// TIA Portal V19 program export: 1 tag tables, 6 data types, 2 data blocks, 8 code blocks (in call order from the OBs), 5 instance data blocks

VAR_GLOBAL   // PLC tag table "Default tag table"
   Tag_1 AT %M0.5 : Bool;
   Clock_Byte AT %MB0 : Byte;
   Clock_10Hz AT %M0.0 : Bool;
   Clock_5Hz AT %M0.1 : Bool;
   "Clock_2.5Hz" AT %M0.2 : Bool;
   Clock_2Hz AT %M0.3 : Bool;
   "Clock_1.25Hz" AT %M0.4 : Bool;
   Clock_1Hz AT %M0.5 : Bool;
   "Clock_0.625Hz" AT %M0.6 : Bool;
   "Clock_0.5Hz" AT %M0.7 : Bool;
   VibSensor01 AT %I100.0 : "PII - BCM R15E-001-DI00-01,5-S4";
   VibSensor02 AT %I124.0 : "PII - BCM R15E-001-DI00-01,5-S4";
   VibSensor03 AT %I148.0 : "PII - BCM R15E-001-DI00-01,5-S4";
   TempHumidSensor01 AT %I172.0 : "PII - CSS 01411.2-xx";
   OilContaminationSensor01 AT %I184.0 : "PII - BCI24-DH367-1D1A-4";
   AirFlowSensor01 AT %I194.0 : "PII - AS5-AF2-FLX-G100";
END_VAR

TYPE "PII - AS5-AF2-FLX-G100"
   STRUCT
      "Process Data In - Mass Flow Rate" : Real;
      "Process Data In - Flow Velocity" : Real;
      "Process Data In - Volume" : Real;
      "Process Data In - Volumetric Flow Rate" : Real;
      "Process Data In - Mass" : Real;
      "Process Data In - Energy" : Real;
      "Process Data In - Temperature" : Real;
      "Process Data In - Pressure" : Real;
      "Port qualifier" : Byte;
   END_STRUCT;
END_TYPE

TYPE "PII - BCI24-DH367-1D1A-4"
   STRUCT
      "Process Data In - Switching output 1" : Bool;
      "Reserved Bit" : Bool;
      "Reserved Bit_1" : Bool;
      "Reserved Bit_2" : Bool;
      "Reserved Bit_3" : Bool;
      "Reserved Bit_4" : Bool;
      "Reserved Bit_5" : Bool;
      "Reserved Bit_6" : Bool;
      "Reserved Byte" : Bool;
      "Process Data In - Pressure" : Word;
      "Reserved Byte_1" : Bool;
      "Reserved Byte_2" : Bool;
      "Reserved Byte_3" : Bool;
      "Reserved Byte_4" : Bool;
      "Reserved Byte_5" : Bool;
      "Reserved Byte_6" : Bool;
      "Reserved Byte_7" : Bool;
      "Reserved Byte_8" : Bool;
      "Reserved Byte_9" : Bool;
      "Reserved Byte_10" : Bool;
      "Reserved Byte_11" : Bool;
      "Reserved Byte_12" : Bool;
      "Reserved Byte_13" : Bool;
      "Reserved Byte_14" : Bool;
      "Reserved Byte_15" : Bool;
      "Reserved Byte_16" : Bool;
      "Reserved Byte_17" : Bool;
      "Reserved Byte_18" : Bool;
      "Reserved Byte_19" : Bool;
      "Reserved Byte_20" : Bool;
      "Reserved Byte_21" : Bool;
      "Reserved Byte_22" : Bool;
      "Reserved Byte_23" : Bool;
      "Reserved Byte_24" : Bool;
      "Reserved Byte_25" : Bool;
      "Reserved Byte_26" : Bool;
      "Reserved Byte_27" : Bool;
      "Reserved Byte_28" : Bool;
      "Port qualifier" : Byte;
   END_STRUCT;
END_TYPE

TYPE "PII - BCM R15E-001-DI00-01,5-S4"
   STRUCT
      "Vibration Acceleration - Vibration Acceleration RMS a-RMS X" : Real;
      "Vibration Acceleration - Vibration Acceleration RMS a-RMS Y" : Real;
      "Vibration Acceleration - Vibration Acceleration RMS a-RMS Z" : Real;
      "Vibration Acceleration - Contact Temperature Contact Temperature" : Real;
      "Vibration Acceleration - Status Bits Main-Alarm a-RMS Magnitude Status" : Bool;
      "Vibration Acceleration - Status Bits Pre-Alarm a-RMS Magnitude Status" : Bool;
      "Vibration Acceleration - Status Bits Main-Alarm a-RMS Z Status" : Bool;
      "Vibration Acceleration - Status Bits Pre-Alarm a-RMS Z Status" : Bool;
      "Vibration Acceleration - Status Bits Main-Alarm a-RMS Y Status" : Bool;
      "Vibration Acceleration - Status Bits Pre-Alarm a-RMS Y Status" : Bool;
      "Vibration Acceleration - Status Bits Main-Alarm a-RMS X Status" : Bool;
      "Vibration Acceleration - Status Bits Pre-Alarm a-RMS X Status" : Bool;
      "Vibration Acceleration - Status Bits Main-Alarm v-RMS Magnitude Status" : Bool;
      "Vibration Acceleration - Status Bits Pre-Alarm v-RMS Magnitude Status" : Bool;
      "Vibration Acceleration - Status Bits Main-Alarm v-RMS Z Status" : Bool;
      "Vibration Acceleration - Status Bits Pre-Alarm v-RMS Z Status" : Bool;
      "Vibration Acceleration - Status Bits Main-Alarm v-RMS Y Status" : Bool;
      "Vibration Acceleration - Status Bits Pre-Alarm v-RMS Y Status" : Bool;
      "Vibration Acceleration - Status Bits Main-Alarm v-RMS X Status" : Bool;
      "Vibration Acceleration - Status Bits Pre-Alarm v-RMS X Status" : Bool;
      "Vibration Acceleration - Status Bits Reserved" : Bool;
      "Vibration Acceleration - Status Bits Reserved_1" : Bool;
      "Vibration Acceleration - Status Bits Reserved_2" : Bool;
      "Vibration Acceleration - Status Bits Vibration Severity Zone D" : Bool;
      "Vibration Acceleration - Status Bits Vibration Severity Zone C" : Bool;
      "Vibration Acceleration - Status Bits Vibration Severity Zone B" : Bool;
      "Vibration Acceleration - Status Bits Vibration Severity Zone A" : Bool;
      "Vibration Acceleration - Status Bits Reserved_3" : Bool;
      "Vibration Acceleration - Status Bits Reserved_4" : Bool;
      "Vibration Acceleration - Status Bits Reserved_5" : Bool;
      "Vibration Acceleration - Status Bits Reserved_6" : Bool;
      "Vibration Acceleration - Status Bits Reserved_7" : Bool;
      "Vibration Acceleration - Status Bits Reserved_8" : Bool;
      "Vibration Acceleration - Status Bits Reserved_9" : Bool;
      "Vibration Acceleration - Status Bits Contact Temperature Upper Alarm Status" : Bool;
      "Vibration Acceleration - Status Bits Contact Temperature Lower Alarm Status" : Bool;
      "Reserved Byte" : Bool;
      "Reserved Byte_1" : Bool;
      "Reserved Byte_2" : Bool;
      "Reserved Byte_3" : Bool;
      "Reserved Byte_4" : Bool;
      "Reserved Byte_5" : Bool;
      "Reserved Byte_6" : Bool;
      "Reserved Byte_7" : Bool;
      "Reserved Byte_8" : Bool;
      "Reserved Byte_9" : Bool;
      "Reserved Byte_10" : Bool;
      "Reserved Byte_11" : Bool;
      "Port qualifier" : Byte;
   END_STRUCT;
END_TYPE

TYPE "PII - CSS 01411.2-xx"
   STRUCT
      "Process Data Inputs - Temperature" : Int;
      "Process Data Inputs - Temperature Alarm High" : Bool;
      "Process Data Inputs - Temperature Range High" : Bool;
      "Process Data Inputs - Temperature Range Low" : Bool;
      "Process Data Inputs - Temperature Alarm Low" : Bool;
      "Reserved Bit" : Bool;
      "Reserved Bit_1" : Bool;
      "Reserved Bit_2" : Bool;
      "Reserved Bit_3" : Bool;
      "Process Data Inputs - Humidity" : Int;
      "Process Data Inputs - Humidity Alarm High" : Bool;
      "Process Data Inputs - Humidity Range High" : Bool;
      "Process Data Inputs - Humidity Range Low" : Bool;
      "Process Data Inputs - Humidity Alarm Low" : Bool;
      "Reserved Bit_4" : Bool;
      "Reserved Bit_5" : Bool;
      "Reserved Bit_6" : Bool;
      "Reserved Bit_7" : Bool;
      "Reserved Byte" : Bool;
      "Reserved Byte_1" : Bool;
      "Reserved Byte_2" : Bool;
      "Reserved Byte_3" : Bool;
      "Reserved Byte_4" : Bool;
      "Reserved Byte_5" : Bool;
      "Reserved Byte_6" : Bool;
      "Reserved Byte_7" : Bool;
      "Reserved Byte_8" : Bool;
      "Reserved Byte_9" : Bool;
      "Reserved Byte_10" : Bool;
      "Reserved Byte_11" : Bool;
      "Reserved Byte_12" : Bool;
      "Reserved Byte_13" : Bool;
      "Reserved Byte_14" : Bool;
      "Reserved Byte_15" : Bool;
      "Reserved Byte_16" : Bool;
      "Reserved Byte_17" : Bool;
      "Reserved Byte_18" : Bool;
      "Reserved Byte_19" : Bool;
      "Reserved Byte_20" : Bool;
      "Reserved Byte_21" : Bool;
      "Reserved Byte_22" : Bool;
      "Reserved Byte_23" : Bool;
      "Reserved Byte_24" : Bool;
      "Reserved Byte_25" : Bool;
      "Port qualifier" : Byte;
   END_STRUCT;
END_TYPE

TYPE "typeSimSensors"
   STRUCT
      Sensors : Struct
         Sensor11 : Real;   // Machine 001 / Sensor 001
         Sensor12 : Real;   // Machine 001 / Sensor 002
         Sensor13 : Real;   // Machine 001 / Sensor 003
         Sensor14 : Real;   // Machine 001 / Sensor 004
         Sensor21 : Real;   // Machine 002 / Sensor 001
         Sensor22 : Real;   // Machine 002 / Sensor 002
         Sensor23 : Real;   // Machine 002 / Sensor 003
         Sensor24 : Real;   // Machine 002 / Sensor 004
      END_STRUCT;
   END_STRUCT;
END_TYPE

TYPE "typeSimStates"
   STRUCT
      States : Struct
         State11 : UInt;   // Machine 1 / State 1
         State12 : UInt;   // Machine 1 / State 2
         State13 : UInt;   // Machine 1 / State 3
         State14 : UInt;   // Machine 1 / State 4
         State21 : UInt;   // Machine 2 / State 1
         State22 : UInt;   // Machine 2 / State 2
         State23 : UInt;   // Machine 2 / State 3
         State24 : UInt;   // Machine 2 / State 4
      END_STRUCT;
   END_STRUCT;
END_TYPE

DATA_BLOCK "GlobalConst_DB"   // DB8
{ S7_Optimized_Access := 'TRUE' }
// stored: MemoryReserve 100
   VAR
      mqtt_host_address : String := '192.168.1.165';
      mqtt_port : UInt := 1883;
      mqtt_username : WString := WSTRING#'mqttbroker';
      mqtt_password : WString := WSTRING#'IoT@2023';
   END_VAR
BEGIN
END_DATA_BLOCK

DATA_BLOCK "GlobalData"   // DB6
{ S7_Optimized_Access := 'TRUE' }
// stored: MemoryReserve 100
   VAR
      UnixTimestamp : DInt;
      SensorsSimulation : "typeSimSensors";
      StatesSimulation { S7_SetPoint := 'True'} : "typeSimStates";
   END_VAR
BEGIN
END_DATA_BLOCK

ORGANIZATION_BLOCK "Main"   // OB1, LAD, ProgramCycle
TITLE = "Main Program Sweep (Cycle)"
{ S7_Optimized_Access := 'TRUE' }
// stored: SetENOAutomatically false
   VAR_INPUT
      Initial_Call : Bool;   // Initial call of this OB
      Remanence : Bool;   // =True, if remanent data are available
   END_VAR
BEGIN

REGION Network 1: Sensor / States simulation
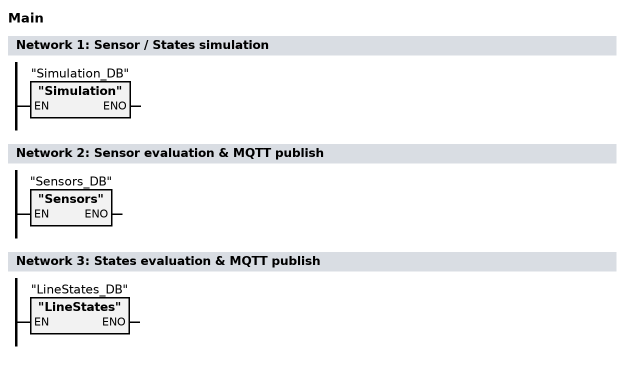
   RUNG wire#powerrail
      "Simulation_DB"()
   END_RUNG
   // the same network as SCL:
   "Simulation_DB"();   // "Simulation"
END_REGION

REGION Network 2: Sensor evaluation & MQTT publish
   RUNG wire#powerrail
      "Sensors_DB"()
   END_RUNG
   // the same network as SCL:
   "Sensors_DB"();   // "Sensors"
END_REGION

REGION Network 3: States evaluation & MQTT publish
   RUNG wire#powerrail
      "LineStates_DB"()
   END_RUNG
   // the same network as SCL:
   "LineStates_DB"();   // "LineStates"
END_REGION
END_ORGANIZATION_BLOCK

FUNCTION_BLOCK "Simulation"   // FB1, LAD
{ S7_Optimized_Access := 'TRUE' }
// stored: MemoryReserve 100, SetENOAutomatically false
   VAR
      LGF_Error : Array[1..10] of Bool;
      LGF_Status : Array[1..10] of Word;
      RetValReal : Real;
   END_VAR
   VAR_TEMP
      RndDIntStatus : Array[1..10] of Word;
      RndRealStatus : Array[1..10] of Word;
   END_VAR
   VAR_TEMP   // added for the SCL form of the ladder/FBD networks
      _w1 : Bool;
      _w2 : Bool;
      _w3 : Bool;
   END_VAR
BEGIN

REGION Network 1: Sensor simulation Machine 1
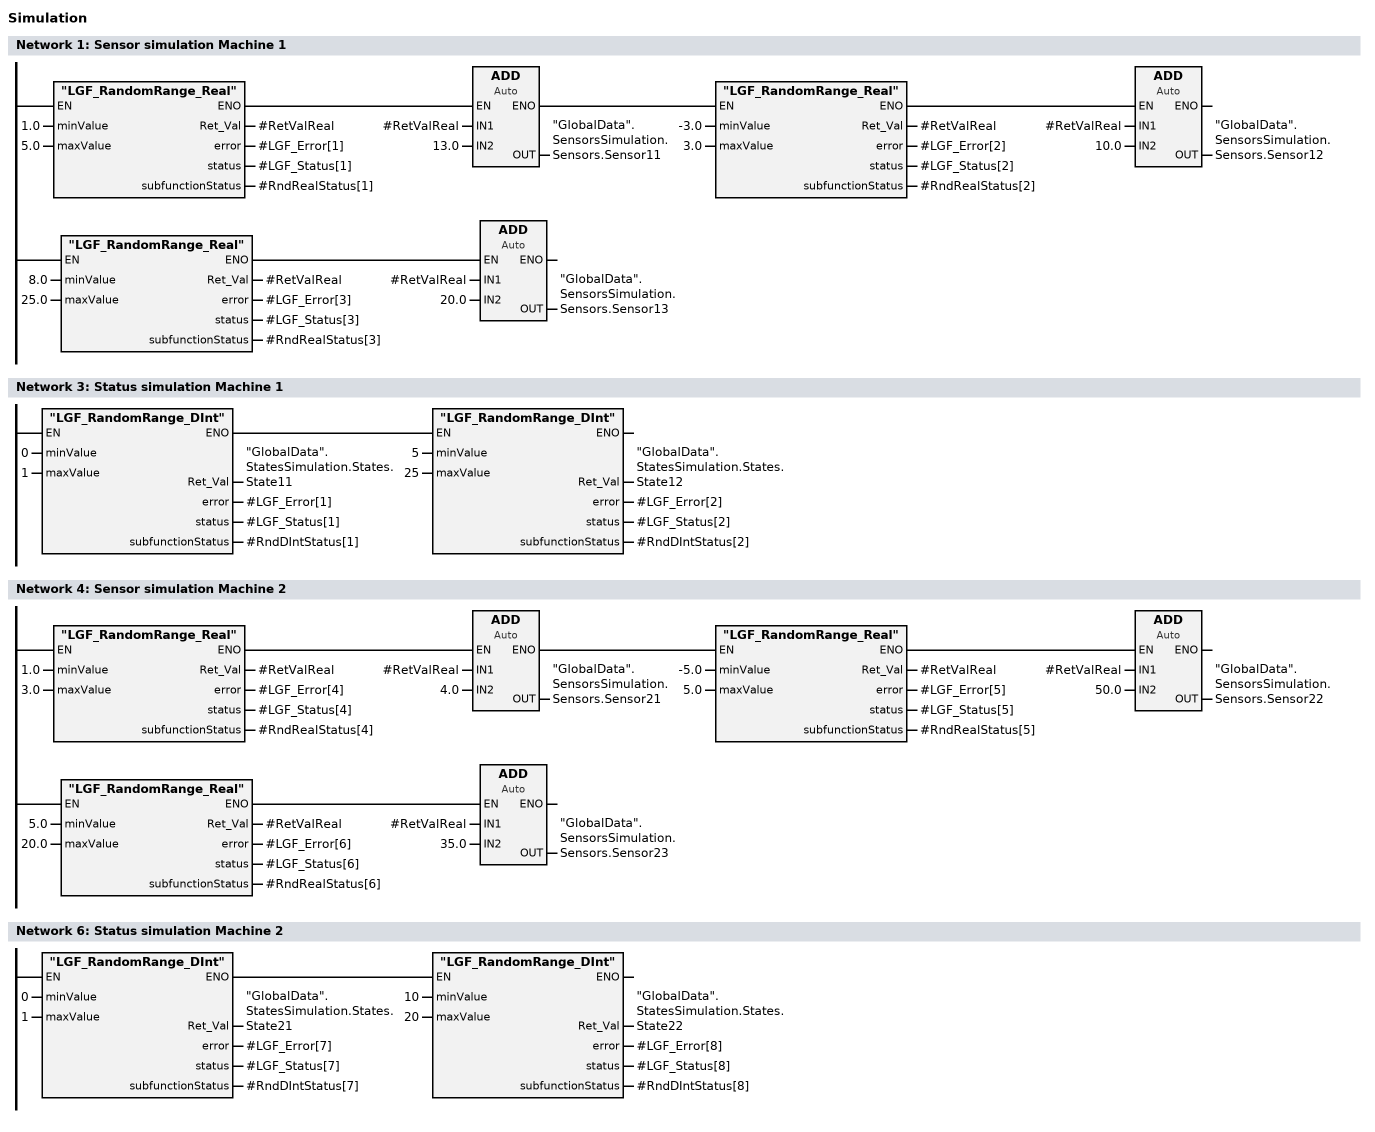
   RUNG wire#powerrail
      "LGF_RandomRange_Real"(minValue := 1.0, maxValue := 5.0, Ret_Val => #RetValReal, error => #LGF_Error[1], status => #LGF_Status[1], subfunctionStatus => #RndRealStatus[1])
      Add(in1 := #RetValReal, in2 := 13.0, out => "GlobalData".SensorsSimulation.Sensors.Sensor11)
      "LGF_RandomRange_Real"(minValue := -3.0, maxValue := 3.0, Ret_Val => #RetValReal, error => #LGF_Error[2], status => #LGF_Status[2], subfunctionStatus => #RndRealStatus[2])
      Add(in1 := #RetValReal, in2 := 10.0, out => "GlobalData".SensorsSimulation.Sensors.Sensor12)
   END_RUNG
   RUNG wire#powerrail
      "LGF_RandomRange_Real"(minValue := 8.0, maxValue := 25.0, Ret_Val => #RetValReal, error => #LGF_Error[3], status => #LGF_Status[3], subfunctionStatus => #RndRealStatus[3])
      Add(in1 := #RetValReal, in2 := 20.0, out => "GlobalData".SensorsSimulation.Sensors.Sensor13)
   END_RUNG
   // the same network as SCL:
   #RetValReal := "LGF_RandomRange_Real"(minValue := 1.0,
                           maxValue := 5.0,
                           error => #LGF_Error[1],
                           status => #LGF_Status[1],
                           subfunctionStatus => #RndRealStatus[1],
                           ENO => #_w1);
   IF #_w1 THEN "GlobalData".SensorsSimulation.Sensors.Sensor11 := #RetValReal + 13.0; END_IF;
   #RetValReal := "LGF_RandomRange_Real"(EN := #_w1,
                           minValue := -3.0,
                           maxValue := 3.0,
                           error => #LGF_Error[2],
                           status => #LGF_Status[2],
                           subfunctionStatus => #RndRealStatus[2],
                           ENO => #_w2);
   IF #_w2 THEN "GlobalData".SensorsSimulation.Sensors.Sensor12 := #RetValReal + 10.0; END_IF;
   #RetValReal := "LGF_RandomRange_Real"(minValue := 8.0,
                           maxValue := 25.0,
                           error => #LGF_Error[3],
                           status => #LGF_Status[3],
                           subfunctionStatus => #RndRealStatus[3],
                           ENO => #_w3);
   IF #_w3 THEN "GlobalData".SensorsSimulation.Sensors.Sensor13 := #RetValReal + 20.0; END_IF;
END_REGION

REGION Network 2 (SCL): Sensor simulation Machine 1
   "GlobalData".SensorsSimulation.Sensors.Sensor14 := "GlobalData".SensorsSimulation.Sensors.Sensor14 + 0.01;

   IF "GlobalData".SensorsSimulation.Sensors.Sensor14 > 100 THEN
       "GlobalData".SensorsSimulation.Sensors.Sensor14 := 0;
   END_IF;
END_REGION

REGION Network 3: Status simulation Machine 1
   RUNG wire#powerrail
      "LGF_RandomRange_DInt"(minValue := 0, maxValue := 1, Ret_Val => "GlobalData".StatesSimulation.States.State11, error => #LGF_Error[1], status => #LGF_Status[1], subfunctionStatus => #RndDIntStatus[1])
      "LGF_RandomRange_DInt"(minValue := 5, maxValue := 25, Ret_Val => "GlobalData".StatesSimulation.States.State12, error => #LGF_Error[2], status => #LGF_Status[2], subfunctionStatus => #RndDIntStatus[2])
   END_RUNG
   // the same network as SCL:
   "GlobalData".StatesSimulation.States.State11 := "LGF_RandomRange_DInt"(minValue := 0,
                           maxValue := 1,
                           error => #LGF_Error[1],
                           status => #LGF_Status[1],
                           subfunctionStatus => #RndDIntStatus[1],
                           ENO => #_w1);
   IF #_w1 THEN
       "GlobalData".StatesSimulation.States.State12 := "LGF_RandomRange_DInt"(minValue := 5,
                               maxValue := 25,
                               error => #LGF_Error[2],
                               status => #LGF_Status[2],
                               subfunctionStatus => #RndDIntStatus[2]);
   END_IF;
END_REGION

REGION Network 4: Sensor simulation Machine 2
   RUNG wire#powerrail
      "LGF_RandomRange_Real"(minValue := 1.0, maxValue := 3.0, Ret_Val => #RetValReal, error => #LGF_Error[4], status => #LGF_Status[4], subfunctionStatus => #RndRealStatus[4])
      Add(in1 := #RetValReal, in2 := 4.0, out => "GlobalData".SensorsSimulation.Sensors.Sensor21)
      "LGF_RandomRange_Real"(minValue := -5.0, maxValue := 5.0, Ret_Val => #RetValReal, error => #LGF_Error[5], status => #LGF_Status[5], subfunctionStatus => #RndRealStatus[5])
      Add(in1 := #RetValReal, in2 := 50.0, out => "GlobalData".SensorsSimulation.Sensors.Sensor22)
   END_RUNG
   RUNG wire#powerrail
      "LGF_RandomRange_Real"(minValue := 5.0, maxValue := 20.0, Ret_Val => #RetValReal, error => #LGF_Error[6], status => #LGF_Status[6], subfunctionStatus => #RndRealStatus[6])
      Add(in1 := #RetValReal, in2 := 35.0, out => "GlobalData".SensorsSimulation.Sensors.Sensor23)
   END_RUNG
   // the same network as SCL:
   #RetValReal := "LGF_RandomRange_Real"(minValue := 1.0,
                           maxValue := 3.0,
                           error => #LGF_Error[4],
                           status => #LGF_Status[4],
                           subfunctionStatus => #RndRealStatus[4],
                           ENO => #_w1);
   IF #_w1 THEN "GlobalData".SensorsSimulation.Sensors.Sensor21 := #RetValReal + 4.0; END_IF;
   #RetValReal := "LGF_RandomRange_Real"(EN := #_w1,
                           minValue := -5.0,
                           maxValue := 5.0,
                           error => #LGF_Error[5],
                           status => #LGF_Status[5],
                           subfunctionStatus => #RndRealStatus[5],
                           ENO => #_w2);
   IF #_w2 THEN "GlobalData".SensorsSimulation.Sensors.Sensor22 := #RetValReal + 50.0; END_IF;
   #RetValReal := "LGF_RandomRange_Real"(minValue := 5.0,
                           maxValue := 20.0,
                           error => #LGF_Error[6],
                           status => #LGF_Status[6],
                           subfunctionStatus => #RndRealStatus[6],
                           ENO => #_w3);
   IF #_w3 THEN "GlobalData".SensorsSimulation.Sensors.Sensor23 := #RetValReal + 35.0; END_IF;
END_REGION

REGION Network 5 (SCL): Sensor simulation Machine 2
   "GlobalData".SensorsSimulation.Sensors.Sensor24 := "GlobalData".SensorsSimulation.Sensors.Sensor24 + 0.1;

   IF "GlobalData".SensorsSimulation.Sensors.Sensor24 > 50 THEN
       "GlobalData".SensorsSimulation.Sensors.Sensor24 := 0;
   END_IF;
END_REGION

REGION Network 6: Status simulation Machine 2
   RUNG wire#powerrail
      "LGF_RandomRange_DInt"(minValue := 0, maxValue := 1, Ret_Val => "GlobalData".StatesSimulation.States.State21, error => #LGF_Error[7], status => #LGF_Status[7], subfunctionStatus => #RndDIntStatus[7])
      "LGF_RandomRange_DInt"(minValue := 10, maxValue := 20, Ret_Val => "GlobalData".StatesSimulation.States.State22, error => #LGF_Error[8], status => #LGF_Status[8], subfunctionStatus => #RndDIntStatus[8])
   END_RUNG
   // the same network as SCL:
   "GlobalData".StatesSimulation.States.State21 := "LGF_RandomRange_DInt"(minValue := 0,
                           maxValue := 1,
                           error => #LGF_Error[7],
                           status => #LGF_Status[7],
                           subfunctionStatus => #RndDIntStatus[7],
                           ENO => #_w1);
   IF #_w1 THEN
       "GlobalData".StatesSimulation.States.State22 := "LGF_RandomRange_DInt"(minValue := 10,
                               maxValue := 20,
                               error => #LGF_Error[8],
                               status => #LGF_Status[8],
                               subfunctionStatus => #RndDIntStatus[8]);
   END_IF;
END_REGION
END_FUNCTION_BLOCK

FUNCTION_BLOCK "Sensors"   // FB4, LAD
{ S7_Optimized_Access := 'TRUE' }
// stored: MemoryReserve 100, SetENOAutomatically false
   VAR
      GenericSensor11 { S7_SetPoint := 'True'} : "GenericSensor";
      GenericSensor12 { S7_SetPoint := 'True'} : "GenericSensor";
      GenericSensor13 { S7_SetPoint := 'True'} : "GenericSensor";
      GenericSensor21 { S7_SetPoint := 'True'} : "GenericSensor";
      GenericSensor22 { S7_SetPoint := 'True'} : "GenericSensor";
      PubJsonMqttInst11 { S7_SetPoint := 'True'} : "PublishJsonMqtt";
      PubJsonMqttInst12 { S7_SetPoint := 'True'} : "PublishJsonMqtt";
      PubJsonMqttInst13 { S7_SetPoint := 'True'} : "PublishJsonMqtt";
      PubJsonMqttInst21 { S7_SetPoint := 'True'} : "PublishJsonMqtt";
      PubJsonMqttInst22 { S7_SetPoint := 'True'} : "PublishJsonMqtt";
      tpGen01 { S7_SetPoint := 'True'} : TP_TIME;
      tpGen02 { S7_SetPoint := 'True'} : TP_TIME;
      tpGen03 { S7_SetPoint := 'True'} : TP_TIME;
      tpGen04 { S7_SetPoint := 'True'} : TP_TIME;
   END_VAR
   VAR_TEMP
      Sensor11 : Real;
      Sensor12 : Real;
      Sensor13 : Real;
      Sensor21 : Real;
      Sensor22 : Real;
   END_VAR
   VAR_TEMP   // added for the SCL form of the ladder/FBD networks
      _w1 : Bool;
   END_VAR
BEGIN

REGION Network 1 (SCL): Generator for data publish Machine 1
   // Define how often sensors are polled and mqtt data sent.
   #tpGen01(IN:=NOT #tpGen02.Q,
            PT:=T#1S);

   #tpGen02(IN:=NOT #tpGen01.Q,
            PT:=T#50MS);
END_REGION

REGION Network 2 (SCL): Generator for data publish Machine 2
   #tpGen03(IN := NOT #tpGen04.Q,
            PT := T#3S);

   #tpGen04(IN := NOT #tpGen03.Q,
            PT := T#50MS);
END_REGION

REGION Network 3: Line 1 / Machine 1 / Sensor 001
   // SELECTOR defines if simulated sensor value or real IO-Link sensor value is evaluated and published by MQTT.
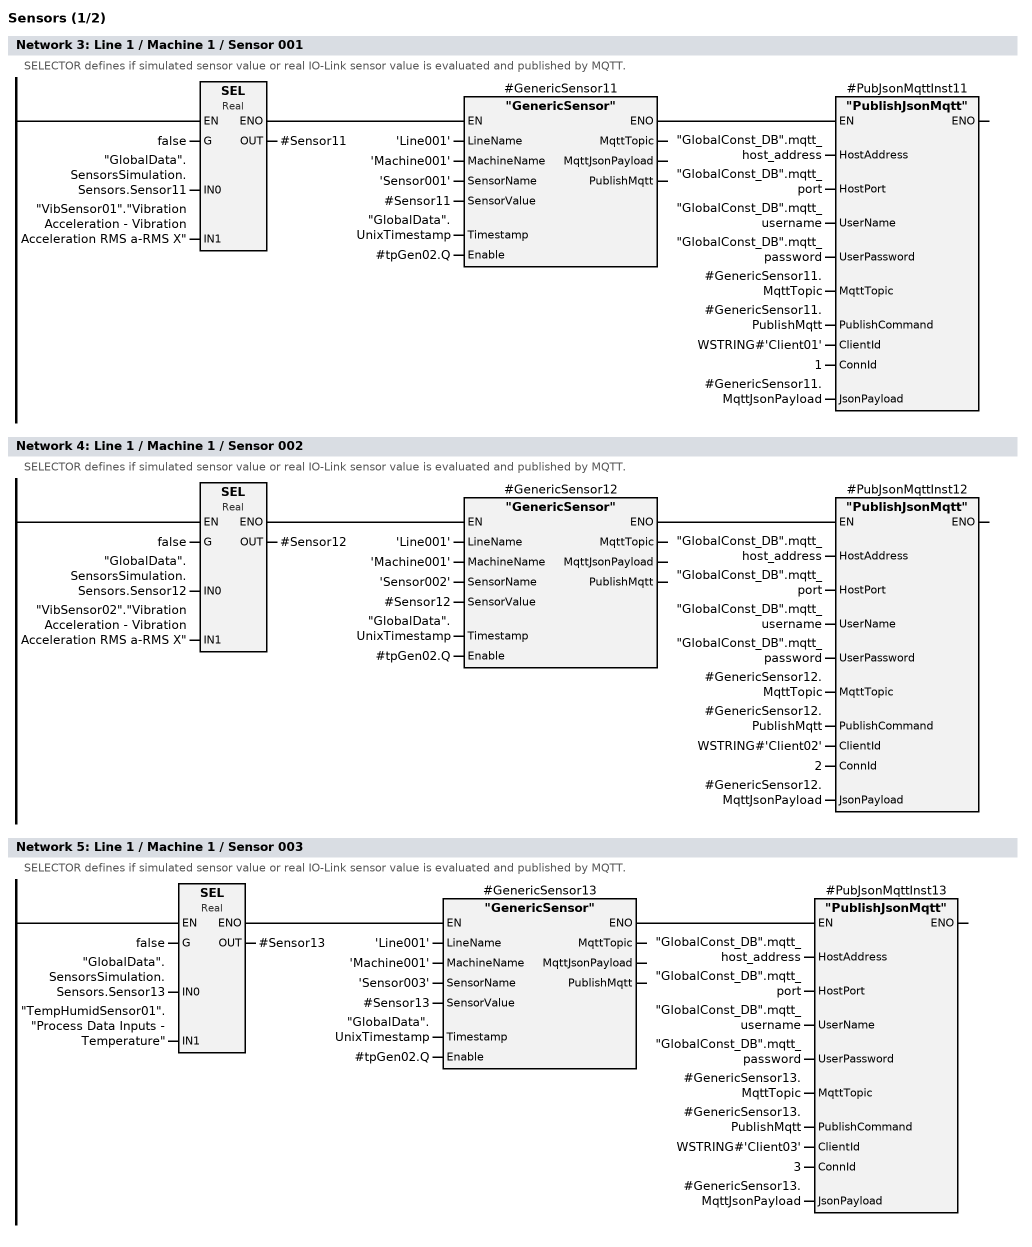
   RUNG wire#powerrail
      { S7_Templates := "value_type := Real" } SEL(g := false, in0 := "GlobalData".SensorsSimulation.Sensors.Sensor11, in1 := "VibSensor01"."Vibration Acceleration - Vibration Acceleration RMS a-RMS X", out => #Sensor11)
      #GenericSensor11(LineName := 'Line001', MachineName := 'Machine001', SensorName := 'Sensor001', SensorValue := #Sensor11, Timestamp := "GlobalData".UnixTimestamp, Enable := #tpGen02.Q, MqttTopic =>, MqttJsonPayload =>, PublishMqtt =>)
      #PubJsonMqttInst11(HostAddress := "GlobalConst_DB".mqtt_host_address, HostPort := "GlobalConst_DB".mqtt_port, UserName := "GlobalConst_DB".mqtt_username, UserPassword := "GlobalConst_DB".mqtt_password, MqttTopic := #GenericSensor11.MqttTopic, PublishCommand := #GenericSensor11.PublishMqtt, ClientId := WSTRING#'Client01', ConnId := 1, JsonPayload := #GenericSensor11.MqttJsonPayload)
   END_RUNG
   // the same network as SCL:
   // ENO of a box is taken as its EN; it also drops when the box reports an error
   #Sensor11 := SEL(G := false, IN0 := "GlobalData".SensorsSimulation.Sensors.Sensor11, IN1 := "VibSensor01"."Vibration Acceleration - Vibration Acceleration RMS a-RMS X");
   #GenericSensor11(LineName := 'Line001',   // "GenericSensor"
                    MachineName := 'Machine001',
                    SensorName := 'Sensor001',
                    SensorValue := #Sensor11,
                    Timestamp := "GlobalData".UnixTimestamp,
                    Enable := #tpGen02.Q,
                    ENO => #_w1);
   IF #_w1 THEN
       #PubJsonMqttInst11(HostAddress := "GlobalConst_DB".mqtt_host_address,   // "PublishJsonMqtt"
                          HostPort := "GlobalConst_DB".mqtt_port,
                          UserName := "GlobalConst_DB".mqtt_username,
                          UserPassword := "GlobalConst_DB".mqtt_password,
                          MqttTopic := #GenericSensor11.MqttTopic,
                          PublishCommand := #GenericSensor11.PublishMqtt,
                          ClientId := WSTRING#'Client01',
                          ConnId := 1,
                          JsonPayload := #GenericSensor11.MqttJsonPayload);
   END_IF;
END_REGION

REGION Network 4: Line 1 / Machine 1 / Sensor 002
   // SELECTOR defines if simulated sensor value or real IO-Link sensor value is evaluated and published by MQTT.
   RUNG wire#powerrail
      { S7_Templates := "value_type := Real" } SEL(g := false, in0 := "GlobalData".SensorsSimulation.Sensors.Sensor12, in1 := "VibSensor02"."Vibration Acceleration - Vibration Acceleration RMS a-RMS X", out => #Sensor12)
      #GenericSensor12(LineName := 'Line001', MachineName := 'Machine001', SensorName := 'Sensor002', SensorValue := #Sensor12, Timestamp := "GlobalData".UnixTimestamp, Enable := #tpGen02.Q, MqttTopic =>, MqttJsonPayload =>, PublishMqtt =>)
      #PubJsonMqttInst12(HostAddress := "GlobalConst_DB".mqtt_host_address, HostPort := "GlobalConst_DB".mqtt_port, UserName := "GlobalConst_DB".mqtt_username, UserPassword := "GlobalConst_DB".mqtt_password, MqttTopic := #GenericSensor12.MqttTopic, PublishCommand := #GenericSensor12.PublishMqtt, ClientId := WSTRING#'Client02', ConnId := 2, JsonPayload := #GenericSensor12.MqttJsonPayload)
   END_RUNG
   // the same network as SCL:
   // ENO of a box is taken as its EN; it also drops when the box reports an error
   #Sensor12 := SEL(G := false, IN0 := "GlobalData".SensorsSimulation.Sensors.Sensor12, IN1 := "VibSensor02"."Vibration Acceleration - Vibration Acceleration RMS a-RMS X");
   #GenericSensor12(LineName := 'Line001',   // "GenericSensor"
                    MachineName := 'Machine001',
                    SensorName := 'Sensor002',
                    SensorValue := #Sensor12,
                    Timestamp := "GlobalData".UnixTimestamp,
                    Enable := #tpGen02.Q,
                    ENO => #_w1);
   IF #_w1 THEN
       #PubJsonMqttInst12(HostAddress := "GlobalConst_DB".mqtt_host_address,   // "PublishJsonMqtt"
                          HostPort := "GlobalConst_DB".mqtt_port,
                          UserName := "GlobalConst_DB".mqtt_username,
                          UserPassword := "GlobalConst_DB".mqtt_password,
                          MqttTopic := #GenericSensor12.MqttTopic,
                          PublishCommand := #GenericSensor12.PublishMqtt,
                          ClientId := WSTRING#'Client02',
                          ConnId := 2,
                          JsonPayload := #GenericSensor12.MqttJsonPayload);
   END_IF;
END_REGION

REGION Network 5: Line 1 / Machine 1 / Sensor 003
   // SELECTOR defines if simulated sensor value or real IO-Link sensor value is evaluated and published by MQTT.
   RUNG wire#powerrail
      { S7_Templates := "value_type := Real" } SEL(g := false, in0 := "GlobalData".SensorsSimulation.Sensors.Sensor13, in1 := "TempHumidSensor01"."Process Data Inputs - Temperature", out => #Sensor13)
      #GenericSensor13(LineName := 'Line001', MachineName := 'Machine001', SensorName := 'Sensor003', SensorValue := #Sensor13, Timestamp := "GlobalData".UnixTimestamp, Enable := #tpGen02.Q, MqttTopic =>, MqttJsonPayload =>, PublishMqtt =>)
      #PubJsonMqttInst13(HostAddress := "GlobalConst_DB".mqtt_host_address, HostPort := "GlobalConst_DB".mqtt_port, UserName := "GlobalConst_DB".mqtt_username, UserPassword := "GlobalConst_DB".mqtt_password, MqttTopic := #GenericSensor13.MqttTopic, PublishCommand := #GenericSensor13.PublishMqtt, ClientId := WSTRING#'Client03', ConnId := 3, JsonPayload := #GenericSensor13.MqttJsonPayload)
   END_RUNG
   // the same network as SCL:
   // ENO of a box is taken as its EN; it also drops when the box reports an error
   #Sensor13 := SEL(G := false, IN0 := "GlobalData".SensorsSimulation.Sensors.Sensor13, IN1 := "TempHumidSensor01"."Process Data Inputs - Temperature");
   #GenericSensor13(LineName := 'Line001',   // "GenericSensor"
                    MachineName := 'Machine001',
                    SensorName := 'Sensor003',
                    SensorValue := #Sensor13,
                    Timestamp := "GlobalData".UnixTimestamp,
                    Enable := #tpGen02.Q,
                    ENO => #_w1);
   IF #_w1 THEN
       #PubJsonMqttInst13(HostAddress := "GlobalConst_DB".mqtt_host_address,   // "PublishJsonMqtt"
                          HostPort := "GlobalConst_DB".mqtt_port,
                          UserName := "GlobalConst_DB".mqtt_username,
                          UserPassword := "GlobalConst_DB".mqtt_password,
                          MqttTopic := #GenericSensor13.MqttTopic,
                          PublishCommand := #GenericSensor13.PublishMqtt,
                          ClientId := WSTRING#'Client03',
                          ConnId := 3,
                          JsonPayload := #GenericSensor13.MqttJsonPayload);
   END_IF;
END_REGION

REGION Network 6: Line 1 / Machine 2 / Sensor 001
   // SELECTOR defines if simulated sensor value or real IO-Link sensor value is evaluated and published by MQTT.
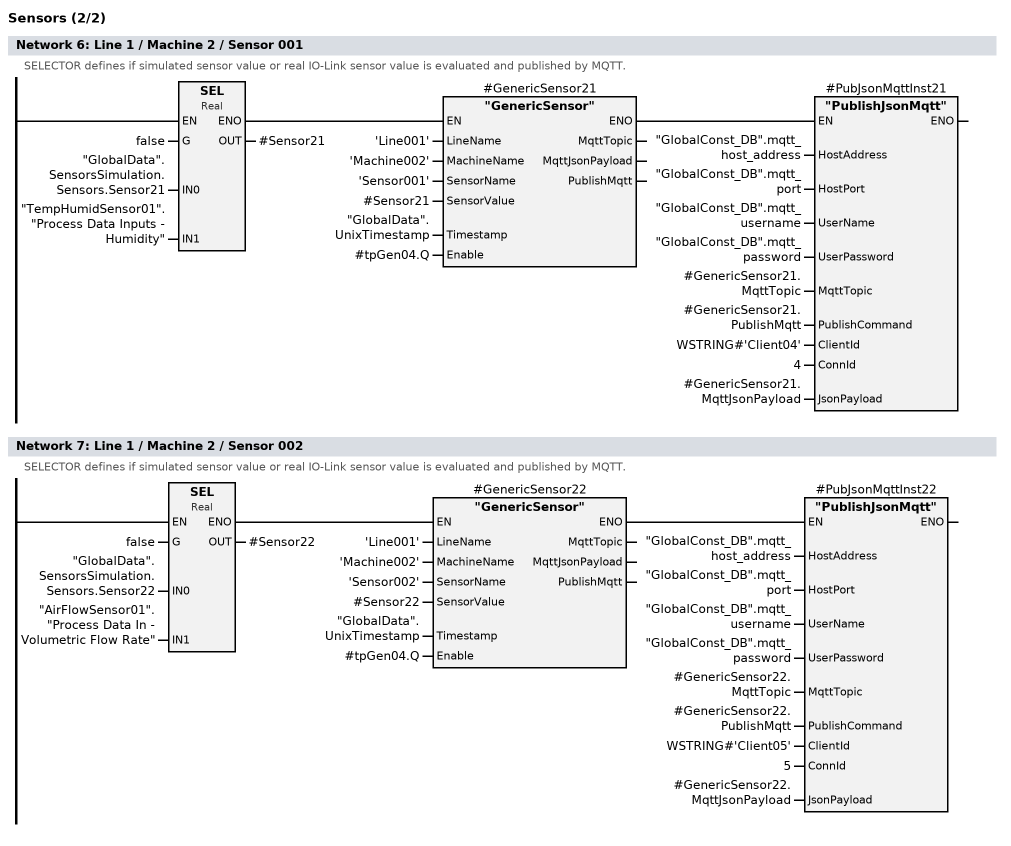
   RUNG wire#powerrail
      { S7_Templates := "value_type := Real" } SEL(g := false, in0 := "GlobalData".SensorsSimulation.Sensors.Sensor21, in1 := "TempHumidSensor01"."Process Data Inputs - Humidity", out => #Sensor21)
      #GenericSensor21(LineName := 'Line001', MachineName := 'Machine002', SensorName := 'Sensor001', SensorValue := #Sensor21, Timestamp := "GlobalData".UnixTimestamp, Enable := #tpGen04.Q, MqttTopic =>, MqttJsonPayload =>, PublishMqtt =>)
      #PubJsonMqttInst21(HostAddress := "GlobalConst_DB".mqtt_host_address, HostPort := "GlobalConst_DB".mqtt_port, UserName := "GlobalConst_DB".mqtt_username, UserPassword := "GlobalConst_DB".mqtt_password, MqttTopic := #GenericSensor21.MqttTopic, PublishCommand := #GenericSensor21.PublishMqtt, ClientId := WSTRING#'Client04', ConnId := 4, JsonPayload := #GenericSensor21.MqttJsonPayload)
   END_RUNG
   // the same network as SCL:
   // ENO of a box is taken as its EN; it also drops when the box reports an error
   #Sensor21 := SEL(G := false, IN0 := "GlobalData".SensorsSimulation.Sensors.Sensor21, IN1 := "TempHumidSensor01"."Process Data Inputs - Humidity");
   #GenericSensor21(LineName := 'Line001',   // "GenericSensor"
                    MachineName := 'Machine002',
                    SensorName := 'Sensor001',
                    SensorValue := #Sensor21,
                    Timestamp := "GlobalData".UnixTimestamp,
                    Enable := #tpGen04.Q,
                    ENO => #_w1);
   IF #_w1 THEN
       #PubJsonMqttInst21(HostAddress := "GlobalConst_DB".mqtt_host_address,   // "PublishJsonMqtt"
                          HostPort := "GlobalConst_DB".mqtt_port,
                          UserName := "GlobalConst_DB".mqtt_username,
                          UserPassword := "GlobalConst_DB".mqtt_password,
                          MqttTopic := #GenericSensor21.MqttTopic,
                          PublishCommand := #GenericSensor21.PublishMqtt,
                          ClientId := WSTRING#'Client04',
                          ConnId := 4,
                          JsonPayload := #GenericSensor21.MqttJsonPayload);
   END_IF;
END_REGION

REGION Network 7: Line 1 / Machine 2 / Sensor 002
   // SELECTOR defines if simulated sensor value or real IO-Link sensor value is evaluated and published by MQTT.
   RUNG wire#powerrail
      { S7_Templates := "value_type := Real" } SEL(g := false, in0 := "GlobalData".SensorsSimulation.Sensors.Sensor22, in1 := "AirFlowSensor01"."Process Data In - Volumetric Flow Rate", out => #Sensor22)
      #GenericSensor22(LineName := 'Line001', MachineName := 'Machine002', SensorName := 'Sensor002', SensorValue := #Sensor22, Timestamp := "GlobalData".UnixTimestamp, Enable := #tpGen04.Q, MqttTopic =>, MqttJsonPayload =>, PublishMqtt =>)
      #PubJsonMqttInst22(HostAddress := "GlobalConst_DB".mqtt_host_address, HostPort := "GlobalConst_DB".mqtt_port, UserName := "GlobalConst_DB".mqtt_username, UserPassword := "GlobalConst_DB".mqtt_password, MqttTopic := #GenericSensor22.MqttTopic, PublishCommand := #GenericSensor22.PublishMqtt, ClientId := WSTRING#'Client05', ConnId := 5, JsonPayload := #GenericSensor22.MqttJsonPayload)
   END_RUNG
   // the same network as SCL:
   // ENO of a box is taken as its EN; it also drops when the box reports an error
   #Sensor22 := SEL(G := false, IN0 := "GlobalData".SensorsSimulation.Sensors.Sensor22, IN1 := "AirFlowSensor01"."Process Data In - Volumetric Flow Rate");
   #GenericSensor22(LineName := 'Line001',   // "GenericSensor"
                    MachineName := 'Machine002',
                    SensorName := 'Sensor002',
                    SensorValue := #Sensor22,
                    Timestamp := "GlobalData".UnixTimestamp,
                    Enable := #tpGen04.Q,
                    ENO => #_w1);
   IF #_w1 THEN
       #PubJsonMqttInst22(HostAddress := "GlobalConst_DB".mqtt_host_address,   // "PublishJsonMqtt"
                          HostPort := "GlobalConst_DB".mqtt_port,
                          UserName := "GlobalConst_DB".mqtt_username,
                          UserPassword := "GlobalConst_DB".mqtt_password,
                          MqttTopic := #GenericSensor22.MqttTopic,
                          PublishCommand := #GenericSensor22.PublishMqtt,
                          ClientId := WSTRING#'Client05',
                          ConnId := 5,
                          JsonPayload := #GenericSensor22.MqttJsonPayload);
   END_IF;
END_REGION
END_FUNCTION_BLOCK

FUNCTION_BLOCK "GenericSensor"
{ S7_Optimized_Access := 'TRUE' }
VERSION : 0.1
   VAR_INPUT 
      LineName : String;
      MachineName : String;
      SensorName : String;
      SensorValue : Real;
      Timestamp : DInt;
      Enable : Bool;
   END_VAR

   VAR_OUTPUT 
      MqttTopic : WString[100];   // mqtt topic
      MqttJsonPayload { ExternalAccessible := 'False'; ExternalVisible := 'False'; ExternalWritable := 'False'} : Array[0..5] of "LStream_typeElement";   // mqtt payload as array of LStream elements
      PublishMqtt : Bool;   // command for publish mqtt payload
   END_VAR

   VAR 
      PayloadSerializedData { ExternalAccessible := 'False'; ExternalVisible := 'False'; ExternalWritable := 'False'; S7_SetPoint := 'False'} : Array[0..5] of "LStream_typeElement" := [(2, 'LineName', (), 0), (2, 'MachineName', (), 0), (2, 'SensorName', (), 0), (3, 'SensorValue', (), 0), (3, 'Timestamp', (), 0), ((), (), (), ())];   // mqtt payload data as serialized LStream elements
      SetParameter { S7_SetPoint := 'True'} : Bool := true;
   END_VAR

   VAR_TEMP 
      TimestampString : String;
      SensorValueString : String;
      TopicString : String;
      RetVal : Int;
      SensorValueInt : Int;
      Size : Int;
   END_VAR


BEGIN
	IF #Enable THEN
	    
	    IF #SetParameter THEN
	        #SetParameter := false;
	        // create mqtt topic
	        #TopicString := CONCAT(IN1 := #LineName, IN2 := #MachineName);
	        #TopicString := INSERT(IN1 := #TopicString, IN2 := '/', P := LEN(#TopicString) - LEN(#MachineName));
	        #TopicString := CONCAT(IN1 := #TopicString, IN2 := #SensorName);
	        #TopicString := INSERT(IN1 := #TopicString, IN2 := '/', P := LEN(#TopicString) - LEN(#SensorName));
	        #MqttTopic := STRING_TO_WSTRING(#TopicString);
	    END_IF;
	    
	    // convert input timestamp to string
	    VAL_STRG(IN := #Timestamp,
	             SIZE := 10,
	             PREC := 0,
	             FORMAT := 0,
	             P := 1,
	             OUT => #TimestampString);
	    
	    #SensorValueInt := REAL_TO_INT(#SensorValue);
	    #SensorValueString := INT_TO_STRING(#SensorValueInt);
	    #Size := LEN(#SensorValueString) + 4;
	    
	    // convert input sensor value to string
	    VAL_STRG(IN := #SensorValue,
	             SIZE := #Size,
	             PREC := 4,
	             FORMAT := 0,
	             P := 1,
	             OUT => #SensorValueString);
	    
	    
	    #PayloadSerializedData[0].value := #LineName;
	    #PayloadSerializedData[1].value := #MachineName;
	    #PayloadSerializedData[2].value := #SensorName;
	    #PayloadSerializedData[3].value := #SensorValueString;
	    #PayloadSerializedData[4].value := #TimestampString;
	    
	    #RetVal := MOVE_BLK_VARIANT(SRC := #PayloadSerializedData,
	                                COUNT := 6,
	                                SRC_INDEX := 0,
	                                DEST_INDEX := 0,
	                                DEST => #MqttJsonPayload);
	    
	    #PublishMqtt := true;
	ELSE
	    #PublishMqtt := false;
	END_IF;
END_FUNCTION_BLOCK

FUNCTION_BLOCK "PublishJsonMqtt"
{ S7_Optimized_Access := 'TRUE' }
VERSION : 0.1
   VAR_INPUT 
      HostAddress : String;
      HostPort : UInt;
      UserName : WString;
      UserPassword : WString[100];
      MqttTopic : WString[100];
      PublishCommand : Bool;
      ClientId : WString;
      ConnId : Word;
   END_VAR

   VAR_IN_OUT 
      JsonPayload : Array[*] of "LStream_typeElement";   // mqtt payload as array of LStream elements
   END_VAR

   VAR 
      MqttClientInstance : "LMQTT_Client";
      SetParameter { S7_SetPoint := 'True'} : Bool := TRUE;
      MqttControl : Struct
         Enable : Bool;
         "Retain" : Bool;
         QoS : Int := 1;
         Publish : Bool;
         Subscribe : Bool;
         Unsubscribe : Bool;
         ConnParam { S7_SetPoint := 'False'} : "LMQTT_typeConnParam" := ((), (), '', 0, (), ());
         ClientId { S7_SetPoint := 'True'} : WString := WSTRING#'';
         User { S7_SetPoint := 'True'} : WString := WSTRING#'';
         Password { S7_SetPoint := 'True'} : WString[500] := WSTRING#'';
         WillTopic : WString;
         WillMsg : Array[0..1023] of Byte;
         Topic : WString[200] := WSTRING#'';
         PublishMsg : Array[0..500] of Byte;
         ReceivedTopic : WString;
         ReceivedMsg : Array[0..999] of Byte;
         ReceivedString : String;
         Valid : Bool;
         Done : Bool;
         Busy : Bool;
         Error : Bool;
         Diagnostic : "typeDiagnostics";
         Status : Word;
         ReceivedMsgStatus : Byte;
         ReceivedMsgDataLen : DWord;
      END_STRUCT;
      LStreamJsonSerializerInst : "LStream_JsonSerializer";
      LStreamSerializer : Struct
         Done : Bool;
         Error : Bool;
         Status : Word;
         ResultCount : UInt;
      END_STRUCT;
      JsonBytePayload : Array[0..500] of Byte;
      rtrigPublishCmd {InstructionName := 'R_TRIG'; LibVersion := '1.0'} : R_TRIG;
   END_VAR

   VAR_TEMP 
      RetVal : Int;
   END_VAR


BEGIN
	IF #SetParameter=TRUE THEN
	    #SetParameter := FALSE;
	    #MqttControl.Topic := #MqttTopic;
	    #MqttControl.ConnParam.broker := #HostAddress;
	    #MqttControl.ConnParam."port" := #HostPort;
	    #MqttControl.ConnParam.connId := #ConnId;
	    #MqttControl.User := #UserName;
	    #MqttControl.Password := #UserPassword;
	    #MqttControl.ClientId := #ClientId;
	END_IF;
	
	#rtrigPublishCmd(CLK:=#PublishCommand);
	
	
	// convert from data objects(array of key-value obejcts) into a compressed JSON data stream (array of bytes)
	#LStreamJsonSerializerInst(execute:=#rtrigPublishCmd.Q ,
	                                 done=>#LStreamSerializer.Done,
	                                 error=>#LStreamSerializer.Error,
	                                 status=>#LStreamSerializer.Status,
	                                 count=>#LStreamSerializer.ResultCount,
	                                 tree:=#JsonPayload,
	                                 jsonByteArray:=#JsonBytePayload);
	
	#MqttControl.PublishMsg := #JsonBytePayload;
	
	// mqtt client instance
	#MqttClientInstance(enable:=true,
	                       publish:=#LStreamSerializer.Done,
	                       subscribe:=false,
	                       unsubscribe:=false,
	                       qos:=1,
	                       retain:=false,
	                       publishMsgLen:=UINT_TO_UDINT(#LStreamSerializer.ResultCount),
	                       willMsgLen:=0,
	                       timeOut:=T#5s,
	                       connParam:=#MqttControl.ConnParam,
	                       clientIdentifier:=#MqttControl.ClientId,
	                       username := #MqttControl.User,
	                       password := #MqttControl.Password,
	                       willtopic:=#MqttControl.WillTopic,
	                       willMsgPayload:=#MqttControl.WillMsg,
	                       mqttTopic:=#MqttTopic,
	                       publishMsgPayload:=#JsonBytePayload,
	                       receivedTopic:=#MqttControl.ReceivedTopic,
	                       receivedMsgPayload:=#MqttControl.ReceivedMsg,
	                       valid=>#MqttControl.Valid,
	                       done=>#MqttControl.Done,
	                       busy=>#MqttControl.Busy,
	                       error=>#MqttControl.Error,
	                       status=>#MqttControl.Status,
	                       diagnostics=>#MqttControl.Diagnostic,
	                       receivedMsgStatus=>#MqttControl.ReceivedMsgStatus,
	                       receivedMsgDataLen=>#MqttControl.ReceivedMsgDataLen
	                        );
	
END_FUNCTION_BLOCK

FUNCTION_BLOCK "LineStates"   // FB8, LAD
{ S7_Optimized_Access := 'TRUE' }
// stored: MemoryReserve 100, SetENOAutomatically false
   VAR
      StateM1LineRunning { S7_SetPoint := 'True'} : "GenericState";
      StateM2LineRunning { S7_SetPoint := 'True'} : "GenericState";
      StateM1CurrentOrderNo { S7_SetPoint := 'True'} : "GenericState";
      StateM2CurrentOrderNo { S7_SetPoint := 'True'} : "GenericState";
      PubJsonMqttInstM1LineRunning { S7_SetPoint := 'True'} : "PublishJsonMqtt";
      PubJsonMqttInstM2LineRunning { S7_SetPoint := 'True'} : "PublishJsonMqtt";
      PubJsonMqttInstM1CurrentOrderNo { S7_SetPoint := 'True'} : "PublishJsonMqtt";
      PubJsonMqttInstM2CurrentOrderNo { S7_SetPoint := 'True'} : "PublishJsonMqtt";
      tpGen01 { S7_SetPoint := 'True'} : TP_TIME;
      tpGen02 { S7_SetPoint := 'True'} : TP_TIME;
   END_VAR
   VAR_TEMP   // added for the SCL form of the ladder/FBD networks
      _w1 : Bool;
   END_VAR
BEGIN

REGION Network 1 (SCL): Generator for data publish
   #tpGen01(IN:=NOT #tpGen02.Q,
            PT:=T#4S);

   #tpGen02(IN:=NOT #tpGen01.Q,
            PT:=T#100MS);
END_REGION

REGION Network 2: Line 1 / Machine 1 / State 'LineRunning'
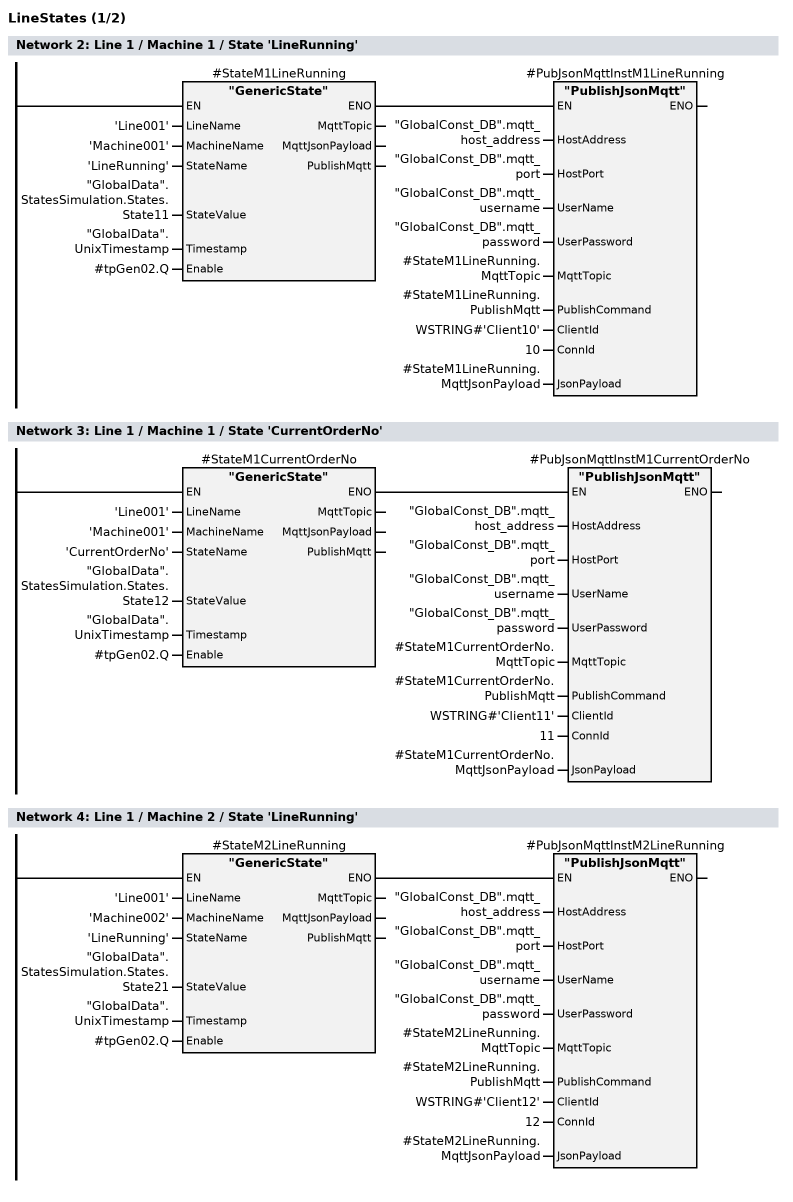
   RUNG wire#powerrail
      #StateM1LineRunning(LineName := 'Line001', MachineName := 'Machine001', StateName := 'LineRunning', StateValue := "GlobalData".StatesSimulation.States.State11, Timestamp := "GlobalData".UnixTimestamp, Enable := #tpGen02.Q, MqttTopic =>, MqttJsonPayload =>, PublishMqtt =>)
      #PubJsonMqttInstM1LineRunning(HostAddress := "GlobalConst_DB".mqtt_host_address, HostPort := "GlobalConst_DB".mqtt_port, UserName := "GlobalConst_DB".mqtt_username, UserPassword := "GlobalConst_DB".mqtt_password, MqttTopic := #StateM1LineRunning.MqttTopic, PublishCommand := #StateM1LineRunning.PublishMqtt, ClientId := WSTRING#'Client10', ConnId := 10, JsonPayload := #StateM1LineRunning.MqttJsonPayload)
   END_RUNG
   // the same network as SCL:
   #StateM1LineRunning(LineName := 'Line001',   // "GenericState"
                       MachineName := 'Machine001',
                       StateName := 'LineRunning',
                       StateValue := "GlobalData".StatesSimulation.States.State11,
                       Timestamp := "GlobalData".UnixTimestamp,
                       Enable := #tpGen02.Q,
                       ENO => #_w1);
   IF #_w1 THEN
       #PubJsonMqttInstM1LineRunning(HostAddress := "GlobalConst_DB".mqtt_host_address,   // "PublishJsonMqtt"
                               HostPort := "GlobalConst_DB".mqtt_port,
                               UserName := "GlobalConst_DB".mqtt_username,
                               UserPassword := "GlobalConst_DB".mqtt_password,
                               MqttTopic := #StateM1LineRunning.MqttTopic,
                               PublishCommand := #StateM1LineRunning.PublishMqtt,
                               ClientId := WSTRING#'Client10',
                               ConnId := 10,
                               JsonPayload := #StateM1LineRunning.MqttJsonPayload);
   END_IF;
END_REGION

REGION Network 3: Line 1 / Machine 1 / State 'CurrentOrderNo'
   RUNG wire#powerrail
      #StateM1CurrentOrderNo(LineName := 'Line001', MachineName := 'Machine001', StateName := 'CurrentOrderNo', StateValue := "GlobalData".StatesSimulation.States.State12, Timestamp := "GlobalData".UnixTimestamp, Enable := #tpGen02.Q, MqttTopic =>, MqttJsonPayload =>, PublishMqtt =>)
      #PubJsonMqttInstM1CurrentOrderNo(HostAddress := "GlobalConst_DB".mqtt_host_address, HostPort := "GlobalConst_DB".mqtt_port, UserName := "GlobalConst_DB".mqtt_username, UserPassword := "GlobalConst_DB".mqtt_password, MqttTopic := #StateM1CurrentOrderNo.MqttTopic, PublishCommand := #StateM1CurrentOrderNo.PublishMqtt, ClientId := WSTRING#'Client11', ConnId := 11, JsonPayload := #StateM1CurrentOrderNo.MqttJsonPayload)
   END_RUNG
   // the same network as SCL:
   #StateM1CurrentOrderNo(LineName := 'Line001',   // "GenericState"
                          MachineName := 'Machine001',
                          StateName := 'CurrentOrderNo',
                          StateValue := "GlobalData".StatesSimulation.States.State12,
                          Timestamp := "GlobalData".UnixTimestamp,
                          Enable := #tpGen02.Q,
                          ENO => #_w1);
   IF #_w1 THEN
       #PubJsonMqttInstM1CurrentOrderNo(HostAddress := "GlobalConst_DB".mqtt_host_address,   // "PublishJsonMqtt"
                               HostPort := "GlobalConst_DB".mqtt_port,
                               UserName := "GlobalConst_DB".mqtt_username,
                               UserPassword := "GlobalConst_DB".mqtt_password,
                               MqttTopic := #StateM1CurrentOrderNo.MqttTopic,
                               PublishCommand := #StateM1CurrentOrderNo.PublishMqtt,
                               ClientId := WSTRING#'Client11',
                               ConnId := 11,
                               JsonPayload := #StateM1CurrentOrderNo.MqttJsonPayload);
   END_IF;
END_REGION

REGION Network 4: Line 1 / Machine 2 / State 'LineRunning'
   RUNG wire#powerrail
      #StateM2LineRunning(LineName := 'Line001', MachineName := 'Machine002', StateName := 'LineRunning', StateValue := "GlobalData".StatesSimulation.States.State21, Timestamp := "GlobalData".UnixTimestamp, Enable := #tpGen02.Q, MqttTopic =>, MqttJsonPayload =>, PublishMqtt =>)
      #PubJsonMqttInstM2LineRunning(HostAddress := "GlobalConst_DB".mqtt_host_address, HostPort := "GlobalConst_DB".mqtt_port, UserName := "GlobalConst_DB".mqtt_username, UserPassword := "GlobalConst_DB".mqtt_password, MqttTopic := #StateM2LineRunning.MqttTopic, PublishCommand := #StateM2LineRunning.PublishMqtt, ClientId := WSTRING#'Client12', ConnId := 12, JsonPayload := #StateM2LineRunning.MqttJsonPayload)
   END_RUNG
   // the same network as SCL:
   #StateM2LineRunning(LineName := 'Line001',   // "GenericState"
                       MachineName := 'Machine002',
                       StateName := 'LineRunning',
                       StateValue := "GlobalData".StatesSimulation.States.State21,
                       Timestamp := "GlobalData".UnixTimestamp,
                       Enable := #tpGen02.Q,
                       ENO => #_w1);
   IF #_w1 THEN
       #PubJsonMqttInstM2LineRunning(HostAddress := "GlobalConst_DB".mqtt_host_address,   // "PublishJsonMqtt"
                               HostPort := "GlobalConst_DB".mqtt_port,
                               UserName := "GlobalConst_DB".mqtt_username,
                               UserPassword := "GlobalConst_DB".mqtt_password,
                               MqttTopic := #StateM2LineRunning.MqttTopic,
                               PublishCommand := #StateM2LineRunning.PublishMqtt,
                               ClientId := WSTRING#'Client12',
                               ConnId := 12,
                               JsonPayload := #StateM2LineRunning.MqttJsonPayload);
   END_IF;
END_REGION

REGION Network 5: Line 1 / Machine 2 / State 'CurrentOrderNo'
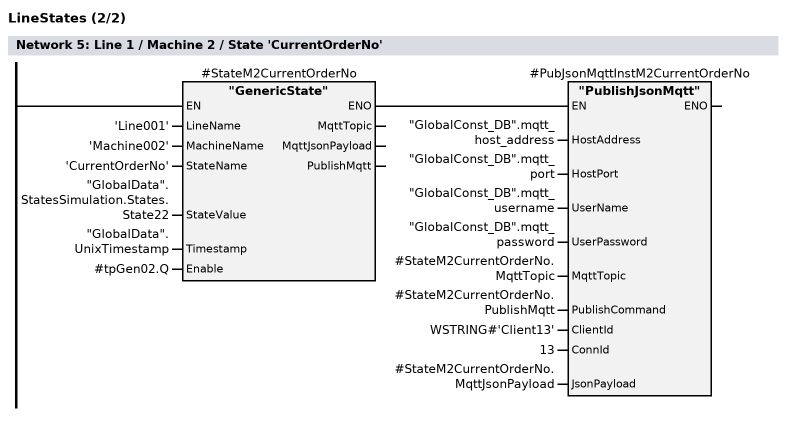
   RUNG wire#powerrail
      #StateM2CurrentOrderNo(LineName := 'Line001', MachineName := 'Machine002', StateName := 'CurrentOrderNo', StateValue := "GlobalData".StatesSimulation.States.State22, Timestamp := "GlobalData".UnixTimestamp, Enable := #tpGen02.Q, MqttTopic =>, MqttJsonPayload =>, PublishMqtt =>)
      #PubJsonMqttInstM2CurrentOrderNo(HostAddress := "GlobalConst_DB".mqtt_host_address, HostPort := "GlobalConst_DB".mqtt_port, UserName := "GlobalConst_DB".mqtt_username, UserPassword := "GlobalConst_DB".mqtt_password, MqttTopic := #StateM2CurrentOrderNo.MqttTopic, PublishCommand := #StateM2CurrentOrderNo.PublishMqtt, ClientId := WSTRING#'Client13', ConnId := 13, JsonPayload := #StateM2CurrentOrderNo.MqttJsonPayload)
   END_RUNG
   // the same network as SCL:
   #StateM2CurrentOrderNo(LineName := 'Line001',   // "GenericState"
                          MachineName := 'Machine002',
                          StateName := 'CurrentOrderNo',
                          StateValue := "GlobalData".StatesSimulation.States.State22,
                          Timestamp := "GlobalData".UnixTimestamp,
                          Enable := #tpGen02.Q,
                          ENO => #_w1);
   IF #_w1 THEN
       #PubJsonMqttInstM2CurrentOrderNo(HostAddress := "GlobalConst_DB".mqtt_host_address,   // "PublishJsonMqtt"
                               HostPort := "GlobalConst_DB".mqtt_port,
                               UserName := "GlobalConst_DB".mqtt_username,
                               UserPassword := "GlobalConst_DB".mqtt_password,
                               MqttTopic := #StateM2CurrentOrderNo.MqttTopic,
                               PublishCommand := #StateM2CurrentOrderNo.PublishMqtt,
                               ClientId := WSTRING#'Client13',
                               ConnId := 13,
                               JsonPayload := #StateM2CurrentOrderNo.MqttJsonPayload);
   END_IF;
END_REGION
END_FUNCTION_BLOCK

FUNCTION_BLOCK "GenericState"
{ S7_Optimized_Access := 'TRUE' }
VERSION : 0.1
   VAR_INPUT 
      LineName : String;
      MachineName : String;
      StateName : String;
      StateValue : UInt;
      Timestamp : DInt;
      Enable : Bool;
   END_VAR

   VAR_OUTPUT 
      MqttTopic : WString[100];   // mqtt topic
      MqttJsonPayload { ExternalAccessible := 'False'; ExternalVisible := 'False'; ExternalWritable := 'False'} : Array[0..5] of "LStream_typeElement";   // mqtt payload as array of LStream elements
      PublishMqtt : Bool;   // command for publish mqtt payload
   END_VAR

   VAR 
      PayloadSerializedData { ExternalAccessible := 'False'; ExternalVisible := 'False'; ExternalWritable := 'False'; S7_SetPoint := 'False'} : Array[0..5] of "LStream_typeElement" := [(2, 'LineName', (), 0), (2, 'MachineName', (), 0), (2, 'StateName', (), 0), (3, 'StateValue', (), 0), (3, 'Timestamp', (), 0), ((), (), (), ())];   // mqtt payload data as serialized LStream elements
      SetParameter { S7_SetPoint := 'True'} : Bool := true;
   END_VAR

   VAR_TEMP 
      TimestampString : String;
      StateValueString : String;
      TopicString : String;
      RetVal : Int;
      SensorValueInt : Int;
      Size : Int;
   END_VAR


BEGIN
	IF #Enable THEN
	    
	    IF #SetParameter THEN
	        #SetParameter := false;
	        // create mqtt topic
	        #TopicString := CONCAT(IN1 := #LineName, IN2 := #MachineName);
	        #TopicString := INSERT(IN1 := #TopicString, IN2 := '/', P := LEN(#TopicString) - LEN(#MachineName));
	        #TopicString := CONCAT(IN1 := #TopicString, IN2 := #StateName);
	        #TopicString := INSERT(IN1 := #TopicString, IN2 := '/', P := LEN(#TopicString) - LEN(#StateName));
	        #MqttTopic := STRING_TO_WSTRING(#TopicString);
	    END_IF;
	    
	    // convert input timestamp to string
	    VAL_STRG(IN := #Timestamp,
	             SIZE := 10,
	             PREC := 0,
	             FORMAT := 0,
	             P := 1,
	             OUT => #TimestampString);
	    
	    #StateValueString := UINT_TO_STRING(#StateValue);
	    #Size := LEN(#StateValueString);
	    
	    // convert input state value to string
	    VAL_STRG(IN := #StateValue,
	             SIZE := #Size,
	             PREC := 0,
	             FORMAT := 0,
	             P := 1,
	             OUT => #StateValueString);
	    
	    
	    #PayloadSerializedData[0].value := #LineName;
	    #PayloadSerializedData[1].value := #MachineName;
	    #PayloadSerializedData[2].value := #StateName;
	    #PayloadSerializedData[3].value := #StateValueString;
	    #PayloadSerializedData[4].value := #TimestampString;
	    
	    #RetVal := MOVE_BLK_VARIANT(SRC := #PayloadSerializedData,
	                                COUNT := 6,
	                                SRC_INDEX := 0,
	                                DEST_INDEX := 0,
	                                DEST => #MqttJsonPayload);
	    
	    #PublishMqtt := true;
	ELSE
	    #PublishMqtt := false;
	END_IF;
END_FUNCTION_BLOCK

ORGANIZATION_BLOCK "TimeStampGenerator"
{ S7_Optimized_Access := 'TRUE' }
VERSION : 0.1
   VAR_TEMP 
      RetVal : Int;
      TimestampDTL {InstructionName := 'DTL'; LibVersion := '1.0'} : DTL;
      UnixTime : DInt;
      UnixTimeError : Bool;
      UnixTimeStatus : Word;
   END_VAR


BEGIN
	// generate Unix timestamp with 1ms resolutionm
	
	#RetVal := RD_LOC_T(#TimestampDTL);
	#UnixTime := "LGF_DTLToUnixTime"(timeDTL := #TimestampDTL,
	                                 error => #UnixTimeError,
	                                 status => #UnixTimeStatus);
	
	"GlobalData".UnixTimestamp := #UnixTime;
END_ORGANIZATION_BLOCK

DATA_BLOCK "LineStates_DB"   // DB9
// stored: InstanceOfName LineStates, InstanceOfType FB
"LineStates"
BEGIN
END_DATA_BLOCK

DATA_BLOCK "Sensors_DB"   // DB4
// stored: InstanceOfName Sensors, InstanceOfType FB
"Sensors"
BEGIN
END_DATA_BLOCK

DATA_BLOCK "Simulation_DB"   // DB7
// stored: InstanceOfName Simulation, InstanceOfType FB
"Simulation"
BEGIN
END_DATA_BLOCK

DATA_BLOCK "LMQTT_Client_DB"   // DB1
AUTHOR : Siemens Industry Online Support
FAMILY : LMQTT
VERSION : 4.0
// stored: InstanceOfName LMQTT_Client, InstanceOfType FB
"LMQTT_Client"
   // VAR_INPUT
   //    enable : Bool;
   //    publish : Bool;
   //    subscribe : Bool;
   //    unsubscribe : Bool;
   //    qos : USInt;
   //    retain : Bool;
   //    publishMsgLen : UDInt;
   //    willMsgLen : UInt;
   //    timeOut : Time;
   // END_VAR
   // VAR_OUTPUT
   //    valid { ExternalWritable := 'False'} : Bool;
   //    done { ExternalWritable := 'False'} : Bool;
   //    busy { ExternalWritable := 'False'} : Bool;
   //    error { ExternalWritable := 'False'} : Bool;
   //    status { ExternalWritable := 'False'} : Word;
   //    diagnostics { ExternalWritable := 'False'} : "typeDiagnostics";
   //    receivedMsgStatus { ExternalWritable := 'False'} : USInt;
   //    receivedMsgDataLen { ExternalWritable := 'False'} : UDInt;
   // END_VAR
   // VAR_IN_OUT
   //    connParam : "LMQTT_typeConnParam";
   //    clientIdentifier : WString;
   //    username : WString;
   //    password : WString;
   //    willtopic : WString;
   //    willMsgPayload : Array[*] of Byte;
   //    mqttTopic : WString;
   //    publishMsgPayload : Array[*] of Byte;
   //    receivedTopic : WString;
   //    receivedMsgPayload : Array[*] of Byte;
   // END_VAR
   // VAR
   //    statEnableOld { ExternalAccessible := 'False'; ExternalVisible := 'False'; ExternalWritable := 'False'} : Bool;
   //    statValid { ExternalAccessible := 'False'; ExternalVisible := 'False'; ExternalWritable := 'False'} : Bool;
   //    statBusy { ExternalAccessible := 'False'; ExternalVisible := 'False'; ExternalWritable := 'False'} : Bool;
   //    statError { ExternalAccessible := 'False'; ExternalVisible := 'False'; ExternalWritable := 'False'} : Bool;
   //    statErrorUserCleared { ExternalAccessible := 'False'; ExternalVisible := 'False'; ExternalWritable := 'False'} : Bool;
   //    statErrorAutoCleared { ExternalAccessible := 'False'; ExternalVisible := 'False'; ExternalWritable := 'False'} : Bool;
   //    statStatus { ExternalAccessible := 'False'; ExternalVisible := 'False'; ExternalWritable := 'False'} : Word;
   //    statDone { ExternalAccessible := 'False'; ExternalVisible := 'False'; ExternalWritable := 'False'} : Bool;
   //    statRcvMsgStatus { ExternalAccessible := 'False'; ExternalVisible := 'False'; ExternalWritable := 'False'} : USInt;
   //    statRcvMsgDataLen { ExternalAccessible := 'False'; ExternalVisible := 'False'; ExternalWritable := 'False'} : UDInt;
   //    statSubfunctionStatus { ExternalAccessible := 'False'; ExternalVisible := 'False'; ExternalWritable := 'False'} : Word;
   //    statFBErrorState { ExternalAccessible := 'False'; ExternalVisible := 'False'; ExternalWritable := 'False'} : DInt;
   //    statFBState { ExternalAccessible := 'False'; ExternalVisible := 'False'; ExternalWritable := 'False'} : DInt;
   //    statMqttConnectState { ExternalAccessible := 'False'; ExternalVisible := 'False'; ExternalWritable := 'False'} : DInt;
   //    statMqttCommandState { ExternalAccessible := 'False'; ExternalVisible := 'False'; ExternalWritable := 'False'} : DInt;
   //    statDisablingCompleted { ExternalAccessible := 'False'; ExternalVisible := 'False'; ExternalWritable := 'False'} : Bool;
   //    statEmptyDiagnostics { ExternalAccessible := 'False'; ExternalVisible := 'False'; ExternalWritable := 'False'} : "typeDiagnostics";
   //    statConnParam { ExternalAccessible := 'False'; ExternalVisible := 'False'; ExternalWritable := 'False'} : Struct
   //       isQDN : Bool;
   //       paramQDN : TCON_QDN_SEC;
   //       paramIP : TCON_IP_V4_SEC;
   //    END_STRUCT;
   //    instTsendC { ExternalAccessible := 'False'; ExternalVisible := 'False'; ExternalWritable := 'False'} : TSEND_C;
   //    instTrcv { ExternalAccessible := 'False'; ExternalVisible := 'False'; ExternalWritable := 'False'} : TRCV;
   //    statSendBuffer { ExternalAccessible := 'False'; ExternalVisible := 'False'; ExternalWritable := 'False'} : Array[0..8191] of Byte;
   //    statRcvBuffer { ExternalAccessible := 'False'; ExternalVisible := 'False'; ExternalWritable := 'False'} : Array[0..1459] of Byte;
   //    statPublishOld { ExternalAccessible := 'False'; ExternalVisible := 'False'; ExternalWritable := 'False'} : Bool;
   //    statSubscribeOld { ExternalAccessible := 'False'; ExternalVisible := 'False'; ExternalWritable := 'False'} : Bool;
   //    statUnsubscribeOld { ExternalAccessible := 'False'; ExternalVisible := 'False'; ExternalWritable := 'False'} : Bool;
   //    statTsendcReq { ExternalAccessible := 'False'; ExternalVisible := 'False'; ExternalWritable := 'False'} : Bool;
   //    statTsendcEnable { ExternalAccessible := 'False'; ExternalVisible := 'False'; ExternalWritable := 'False'} : Bool;
   //    statTsendcLen { ExternalAccessible := 'False'; ExternalVisible := 'False'; ExternalWritable := 'False'} : UDInt;
   //    statEnableTimerCommandWatchdog { ExternalAccessible := 'False'; ExternalVisible := 'False'; ExternalWritable := 'False'} : Bool;
   //    instTimerCommandWatchdog { ExternalAccessible := 'False'; ExternalVisible := 'False'; ExternalWritable := 'False'} : IEC_TIMER;
   //    statEnableMqttKeepAliveTimer { ExternalAccessible := 'False'; ExternalVisible := 'False'; ExternalWritable := 'False'} : Bool;
   //    statMqttKeepAliveUsed { ExternalAccessible := 'False'; ExternalVisible := 'False'; ExternalWritable := 'False'} : Bool;
   //    statMqttKeepAliveTime { ExternalAccessible := 'False'; ExternalVisible := 'False'; ExternalWritable := 'False'} : Time;
   //    instMqttKeepAliveTimer { ExternalAccessible := 'False'; ExternalVisible := 'False'; ExternalWritable := 'False'} : IEC_TIMER;
   //    statSendBufferPos { ExternalAccessible := 'False'; ExternalVisible := 'False'; ExternalWritable := 'False'} : UInt;
   //    statPaketHeaderEncodeDone { ExternalAccessible := 'False'; ExternalVisible := 'False'; ExternalWritable := 'False'} : Bool;
   //    statSendPaketTotalRemLen { ExternalAccessible := 'False'; ExternalVisible := 'False'; ExternalWritable := 'False'} : UDInt;
   //    statEncodedRemPaketLenAsByte { ExternalAccessible := 'False'; ExternalVisible := 'False'; ExternalWritable := 'False'} : Byte;
   //    statUsernameLenUtf8Encoded { ExternalAccessible := 'False'; ExternalVisible := 'False'; ExternalWritable := 'False'} : UInt;
   //    statPasswordLenUtf8Encoded { ExternalAccessible := 'False'; ExternalVisible := 'False'; ExternalWritable := 'False'} : UInt;
   //    statWillTopicLenUtf8Encoded { ExternalAccessible := 'False'; ExternalVisible := 'False'; ExternalWritable := 'False'} : UInt;
   //    statClientIdLenUtf8Encoded { ExternalAccessible := 'False'; ExternalVisible := 'False'; ExternalWritable := 'False'} : UInt;
   //    statWillQos { ExternalAccessible := 'False'; ExternalVisible := 'False'; ExternalWritable := 'False'} : USInt;
   //    statWillRetain { ExternalAccessible := 'False'; ExternalVisible := 'False'; ExternalWritable := 'False'} : Bool;
   //    statWillMessageCnt { ExternalAccessible := 'False'; ExternalVisible := 'False'; ExternalWritable := 'False'} : UInt;
   //    statClientIdPos { ExternalAccessible := 'False'; ExternalVisible := 'False'; ExternalWritable := 'False'} : DInt;
   //    statClientIdEncodeState { ExternalAccessible := 'False'; ExternalVisible := 'False'; ExternalWritable := 'False'} : DInt;
   //    statWillMessagePos { ExternalAccessible := 'False'; ExternalVisible := 'False'; ExternalWritable := 'False'} : DInt;
   //    statWillMessageEncodeState { ExternalAccessible := 'False'; ExternalVisible := 'False'; ExternalWritable := 'False'} : DInt;
   //    statWillTopicPos { ExternalAccessible := 'False'; ExternalVisible := 'False'; ExternalWritable := 'False'} : DInt;
   //    statWillTopicEncodeState { ExternalAccessible := 'False'; ExternalVisible := 'False'; ExternalWritable := 'False'} : DInt;
   //    statUserNamePos { ExternalAccessible := 'False'; ExternalVisible := 'False'; ExternalWritable := 'False'} : DInt;
   //    statUserNameEncodeState { ExternalAccessible := 'False'; ExternalVisible := 'False'; ExternalWritable := 'False'} : DInt;
   //    statPasswordPos { ExternalAccessible := 'False'; ExternalVisible := 'False'; ExternalWritable := 'False'} : DInt;
   //    statPasswordEncodeState { ExternalAccessible := 'False'; ExternalVisible := 'False'; ExternalWritable := 'False'} : DInt;
   //    statPaketId { ExternalAccessible := 'False'; ExternalVisible := 'False'; ExternalWritable := 'False'} : UInt;
   //    statPublishTopicLenUtf8Encoded { ExternalAccessible := 'False'; ExternalVisible := 'False'; ExternalWritable := 'False'} : UInt;
   //    statPublishQos { ExternalAccessible := 'False'; ExternalVisible := 'False'; ExternalWritable := 'False'} : USInt;
   //    statPublishMessageCnt { ExternalAccessible := 'False'; ExternalVisible := 'False'; ExternalWritable := 'False'} : UDInt;
   //    statPublishTopicEncodeState { ExternalAccessible := 'False'; ExternalVisible := 'False'; ExternalWritable := 'False'} : DInt;
   //    statPublishTopicPos { ExternalAccessible := 'False'; ExternalVisible := 'False'; ExternalWritable := 'False'} : DInt;
   //    statPaketIdEncoded { ExternalAccessible := 'False'; ExternalVisible := 'False'; ExternalWritable := 'False'} : Bool;
   //    statPublishEncodeMessageState { ExternalAccessible := 'False'; ExternalVisible := 'False'; ExternalWritable := 'False'} : DInt;
   //    statPublishMessagePos { ExternalAccessible := 'False'; ExternalVisible := 'False'; ExternalWritable := 'False'} : DInt;
   //    statSubscribeQos { ExternalAccessible := 'False'; ExternalVisible := 'False'; ExternalWritable := 'False'} : USInt;
   //    statSubscribeQosEncoded { ExternalAccessible := 'False'; ExternalVisible := 'False'; ExternalWritable := 'False'} : Bool;
   //    statSubscribeTopicPos { ExternalAccessible := 'False'; ExternalVisible := 'False'; ExternalWritable := 'False'} : DInt;
   //    statSubscribeTopicEncodeState { ExternalAccessible := 'False'; ExternalVisible := 'False'; ExternalWritable := 'False'} : DInt;
   //    statSubscribeTopicLenUtf8Encoded { ExternalAccessible := 'False'; ExternalVisible := 'False'; ExternalWritable := 'False'} : UInt;
   //    statUnsubscribeTopicPos { ExternalAccessible := 'False'; ExternalVisible := 'False'; ExternalWritable := 'False'} : DInt;
   //    statUnsubscribeTopicEncodeState { ExternalAccessible := 'False'; ExternalVisible := 'False'; ExternalWritable := 'False'} : DInt;
   //    statUnsubscribeTopicLenUtf8Encoded { ExternalAccessible := 'False'; ExternalVisible := 'False'; ExternalWritable := 'False'} : UInt;
   //    statRcvMsgQoS { ExternalAccessible := 'False'; ExternalVisible := 'False'; ExternalWritable := 'False'} : UInt;
   //    statRcvMsgTotalLen { ExternalAccessible := 'False'; ExternalVisible := 'False'; ExternalWritable := 'False'} : UDInt;
   //    statRcvMsgTopicLen { ExternalAccessible := 'False'; ExternalVisible := 'False'; ExternalWritable := 'False'} : UInt;
   //    statRcvMsgPayloadLen { ExternalAccessible := 'False'; ExternalVisible := 'False'; ExternalWritable := 'False'} : UDInt;
   //    statRcvMsgPaketId { ExternalAccessible := 'False'; ExternalVisible := 'False'; ExternalWritable := 'False'} : Word;
   //    statRcvMsgTopicPos { ExternalAccessible := 'False'; ExternalVisible := 'False'; ExternalWritable := 'False'} : DInt;
   //    statRcvMsgPayloadPos { ExternalAccessible := 'False'; ExternalVisible := 'False'; ExternalWritable := 'False'} : DInt;
   //    statRcvMsgDecodeState { ExternalAccessible := 'False'; ExternalVisible := 'False'; ExternalWritable := 'False'} : DInt;
   //    statRcvMsgInternalStatus { ExternalAccessible := 'False'; ExternalVisible := 'False'; ExternalWritable := 'False'} : USInt;
   //    statMqttPubRecRcv { ExternalAccessible := 'False'; ExternalVisible := 'False'; ExternalWritable := 'False'} : USInt;
   //    statSendPubAckMsg { ExternalAccessible := 'False'; ExternalVisible := 'False'; ExternalWritable := 'False'} : Bool;
   //    statPubRecReady { ExternalAccessible := 'False'; ExternalVisible := 'False'; ExternalWritable := 'False'} : Bool;
   //    statCommandInputOld { ExternalAccessible := 'False'; ExternalVisible := 'False'; ExternalWritable := 'False'} : Bool;
   //    statCommandInputBackup { ExternalAccessible := 'False'; ExternalVisible := 'False'; ExternalWritable := 'False'} : Byte;
   // END_VAR
BEGIN
END_DATA_BLOCK

DATA_BLOCK "LStream_JsonSerializer_DB"   // DB2
AUTHOR : DI_FA_S_SUP_EuC
FAMILY : LStream
VERSION : 1.0
// stored: InstanceOfName LStream_JsonSerializer, InstanceOfType FB
"LStream_JsonSerializer"
   // VAR_INPUT
   //    execute { ExternalAccessible := 'False'; ExternalVisible := 'False'; ExternalWritable := 'False'} : Bool;
   // END_VAR
   // VAR_OUTPUT
   //    done { ExternalAccessible := 'False'; ExternalVisible := 'False'; ExternalWritable := 'False'} : Bool;
   //    busy { ExternalAccessible := 'False'; ExternalVisible := 'False'; ExternalWritable := 'False'} : Bool;
   //    error { ExternalAccessible := 'False'; ExternalVisible := 'False'; ExternalWritable := 'False'} : Bool;
   //    status { ExternalAccessible := 'False'; ExternalVisible := 'False'; ExternalWritable := 'False'} : Word;
   //    count { ExternalAccessible := 'False'; ExternalVisible := 'False'; ExternalWritable := 'False'} : UInt;
   // END_VAR
   // VAR_IN_OUT
   //    tree : Array[*] of "LStream_typeElement";
   //    jsonByteArray : Array[*] of Byte;
   // END_VAR
   // VAR
   //    statExecuteOld { ExternalAccessible := 'False'; ExternalVisible := 'False'; ExternalWritable := 'False'} : Bool;
   //    statDone { ExternalAccessible := 'False'; ExternalVisible := 'False'; ExternalWritable := 'False'} : Bool;
   //    statBusy { ExternalAccessible := 'False'; ExternalVisible := 'False'; ExternalWritable := 'False'} : Bool;
   //    statError { ExternalAccessible := 'False'; ExternalVisible := 'False'; ExternalWritable := 'False'} : Bool;
   //    statCount { ExternalAccessible := 'False'; ExternalVisible := 'False'; ExternalWritable := 'False'} : UInt;
   //    statStatus { ExternalAccessible := 'False'; ExternalVisible := 'False'; ExternalWritable := 'False'} : Word;
   //    statFbState { ExternalAccessible := 'False'; ExternalVisible := 'False'; ExternalWritable := 'False'} : DInt;
   //    statFbPreviousState { ExternalAccessible := 'False'; ExternalVisible := 'False'; ExternalWritable := 'False'} : DInt;
   //    statFbNextState { ExternalAccessible := 'False'; ExternalVisible := 'False'; ExternalWritable := 'False'} : DInt;
   //    statIndexJsonByteArray { ExternalAccessible := 'False'; ExternalVisible := 'False'; ExternalWritable := 'False'} : UInt;
   //    statIndexTreeArray { ExternalAccessible := 'False'; ExternalVisible := 'False'; ExternalWritable := 'False'} : UInt;
   //    statTreeLen { ExternalAccessible := 'False'; ExternalVisible := 'False'; ExternalWritable := 'False'} : DInt;
   //    statJsonByteLen { ExternalAccessible := 'False'; ExternalVisible := 'False'; ExternalWritable := 'False'} : DInt;
   //    statInfoToWrite { ExternalAccessible := 'False'; ExternalVisible := 'False'; ExternalWritable := 'False'} : String;
   //    statIsLastElement { ExternalAccessible := 'False'; ExternalVisible := 'False'; ExternalWritable := 'False'} : Bool;
   //    statLastElementIsClosed { ExternalAccessible := 'False'; ExternalVisible := 'False'; ExternalWritable := 'False'} : Bool;
   //    statStackIndexOpenElement { ExternalAccessible := 'False'; ExternalVisible := 'False'; ExternalWritable := 'False'} : Array[0..10] of Char;
   //    statStackIndex { ExternalAccessible := 'False'; ExternalVisible := 'False'; ExternalWritable := 'False'} : Int;
   //    instWatchdog { ExternalAccessible := 'False'; ExternalVisible := 'False'; ExternalWritable := 'False'} : IEC_TIMER;
   //    statIsArrayOpen : Bool;
   //    statIsArrayFieldClosed : Bool;
   //    statIsFirstElement : Bool;
   //    statFirstArrayKey : String;
   //    statArrayName : String;
   // END_VAR
BEGIN
END_DATA_BLOCK
